INTERFACE I_Cylinder

METHOD PUBLIC FullyExtend
VAR_INPUT
END_VAR
END_METHOD

METHOD PUBLIC FullyRetract
VAR_INPUT
END_VAR
END_METHOD

PROPERTY PUBLIC IsFullyExtended : BOOL
GET
END_GET
END_PROPERTY

PROPERTY PUBLIC IsFullyRetracted : BOOL
GET
END_GET
END_PROPERTY

END_INTERFACE

(* stored: Version 1.1.0.1, ProductVersion 3.1.4024.11
   Itf I_Cylinder: Id {cac00173-be50-43e3-880c-78a937c8884e}
   Method FullyExtend: Id {328cf513-3d82-4b44-9cf5-1304a3e5a36b}
   Method FullyRetract: Id {b937f871-631f-42a9-8abc-fb05ae02a571}
   Property IsFullyExtended: Id {9c0850e5-eb39-4184-a5da-c4666a78dd97}
   Get Get: Id {0c1ae2d2-cdd9-4361-8758-82d5902ed66e}
   Property IsFullyRetracted: Id {7a4c7535-b029-4fed-a6be-79f5ffbd4dcb}
   Get Get: Id {93b1d24e-6565-40b6-bd53-8c337b335014} *)
